(* PLC project v0.6.02_RefactorGateAndTest.project, CODESYS CODESYS V3.5 SP19 Patch 1 *)
(* stored: creationDateTime 2026-08-14T10:10:49.359610, modificationDateTime 2026-08-14T10:10:49.359610 *)

(* ═══════════════════════════════════════════════════════════════ 🔧 ST_CommunCfg — Configuration des paramètres communs machine 📄 2026-07-24 : WinchMaxStepDescente/WinchMaxStepAscent/WinchSlowdownDistance_M/ WinchSlowSpeed_Pct rapatriés depuis ST_WinchCfg (étaient partagés M1/M2 par réconciliation ad-hoc dans PRG_SUPERVISION_CFC.st, une seule instance ici l'élimine). ═══════════════════════════════════════════════════════════════ *)
TYPE ST_CommunCfg : STRUCT
  LimitLegalDepthMinAllowed_M : REAL := -999;  (* 🔴🔧 REX 2026-08-07 (5) — retour terrain, blocage instantané à 0m : sans défaut explicite, ce champ vaut 0.0 tant qu'il n'a pas été réglé côté IHM -- "CablePosM <= 0.0" se déclenche dès la position de référence, avant tout réglage réel de la cote légale. Défaut -999.0 (jamais atteint en pratique) : LimitLegalEnabled=TRUE sans réglage ne bloque plus rien par erreur -- il faut régler la vraie cote pour que la protection devienne active. 📐 Cote min de dragage autorisée (m, négatif) *)
  LimitLegalEnabled : BOOL;  (* 🟢 Activation de la limite légale *)
  SelHomingApproachEnable : BOOL;  (* 🔌 Case IHM : autorise le dépassement butée haute pour homing (si MAINT_N2) *)
  WinchMaxStepDescente : INT := 3;  (* 🛑 Limitation palier vitesse en descente (1..5), commun M1/M2 *)
  WinchMaxStepAscent : INT := 5;  (* 🚀 Limitation palier vitesse en montée (1..5), commun M1/M2 *)
  WinchSlowdownDistance_M : REAL := 1;  (* 📏 Distance avant limite pour enclencher le ralentissement (m), commun M1/M2 *)
  WinchSlowdownMaxStep : INT := 1;  (* 🔧 2026-08-07 : WinchSlowSpeed_Pct (%) retiré — un treuil ne connaît que des paliers (1..5), pas une vitesse continue. 🆕 2026-08-07 : Plafond palier dans la zone de ralentissement (1..5), commun M1/M2 *)
  TglEnableKoboldAutoStopDescent : BOOL := FALSE;  (* 🆕 2026-08-07 : Arrêt auto descente sur détection fond Kobold (pilotage normal) *)
  TglEnableCoupledBucketSequencing : BOOL := FALSE;  (* 🔴🔧 REX 2026-08-07 (4) — coupe-circuit d'urgence pour le séquencement auto benne (Fiche 01). Défaut FALSE = comportement IDENTIQUE à avant Fiche 01 (déplacement M1/M2 synchro jamais gouverné par instBucket.Busy sauf action MANUELLE benne/DumpAtTremie/ExtractionSequence). *)
  Initialized : BOOL := FALSE;  (* 🚦 flag restauration boot *)
END_STRUCT;
END_TYPE

(* ═══════════════════════════════════════════════════════════════ 🌉 FB_CfgPersistBridge_CommunCfg — Pont persistance générique pour ST_CommunCfg ─────────────────────────────────────────────────────────────── 🎯 Voir FB_CfgPersistBridge_SyncCfg.st (Lot 3a) pour la logique de référence — identique, seul le type ST_CommunCfg change. ═══════════════════════════════════════════════════════════════ *)
FUNCTION_BLOCK FB_CfgPersistBridge_CommunCfg
  VAR_OUTPUT
    JustRestored : BOOL;
  END_VAR
  VAR_IN_OUT
    Hmi : ST_CommunCfg;  (* 🖥️ ex. GVL_IHM.Commun.Cfg *)
    Persist : ST_CommunCfg;  (* 💾 ex. GVL_PERSISTENT._CommunCfgPersist *)
  END_VAR

            

JustRestored := FALSE;
IF NOT Hmi.Initialized THEN
    Hmi := Persist;
    Hmi.Initialized := TRUE;
    JustRestored := TRUE;
ELSE
    Persist := Hmi;
END_IF;

          
END_FUNCTION_BLOCK
